// TIA Portal project "LampModel" (V16)

(* hardware
DEVICE "HMI_1"  TP700 Comfort
   slot 0: "HMI_1"  TP700 Comfort  6AV2 124-0GC01-0AX0  16.0.0.0
   slot 1: "HMI_RT_1"  TP700 Comfort  6AV2 124-0GC01-0AX0  16.0.0.0
   slot 5: "HMI_1.IE_CP_1"  PROFINET Interface  16.0.0.0
      slot 1: "PROFINET Interface_1"  PROFINET Interface
         slot 1: "Port_1"  Port
         slot 2: "Port_2"  Port
   slot 7: "HMI_1.MPI/DP_CP_1"  MPI/DP Interface  16.0.0.0
DEVICE "S71500/ET200MP station_1"  S7-1500 station
   slot 0: "Rail_0"  Rack  6ES7 590-1***0-0AA0
   slot 1: "PLC_1"  CPU 1518-4 PN/DP  6ES7 518-4AP00-0AB0  V2.8
      slot 3: "CPU display_1"  6ES7591-1BA00-0AA0
      slot 32768: "PROFINET interface_1"  X1
         slot 32769: "Port_1"  X1 P1
         slot 32770: "Port_2"  X1 P2
      slot 33024: "PROFINET interface_2"  X2
         slot 33025: "Port_1"  X2 P1
      slot 33280: "PROFINET interface GBIT_3"  X3
         slot 33281: "Port_1"  X3 P1
      slot 33536: "DP interface_1"  X4
      slot 34817: "Virtual CP interface port_1"  Virtual CP interface port  Virtual CP interface port
*)

// ===== PLC "PLC_1"  CPU 1518-4 PN/DP =====

VAR_GLOBAL   // PLC tag table "Default tag table"
   "Lambayı Yak" AT %M0.0 : Bool;
   "Lamba" AT %M0.1 : Bool;
   "PTRIG" AT %M0.2 : Bool;
   "PTRIG1" AT %M0.3 : Bool;
   "NTRIG" AT %M0.4 : Bool;
   "PTRIG3" AT %M0.5 : Bool;
   "ntrıg2" AT %M0.6 : Bool;
END_VAR

ORGANIZATION_BLOCK "Main"   // OB1, LAD, ProgramCycle
TITLE = "Main Program Sweep (Cycle)"
{ S7_Optimized_Access := 'TRUE' }
VERSION : 0.1
   VAR_INPUT
      Initial_Call : Bool;   // Initial call of this OB
      Remanence : Bool;   // =True, if remanent data are available
   END_VAR
   VAR_TEMP   // added for the SCL form of the ladder/FBD networks
      _w1 : Bool;
      _w2 : Bool;
   END_VAR
BEGIN

REGION Network 1
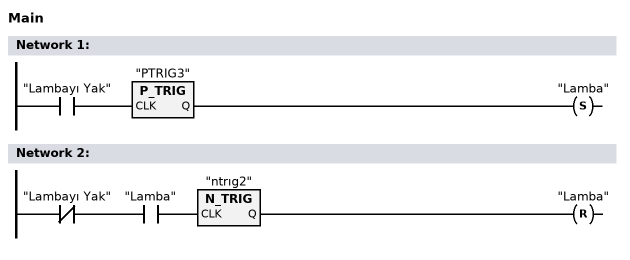
   RUNG wire#powerrail
      Contact( "Lambayı Yak" )
      P_Trig( "PTRIG3" )
      S_Coil( "Lamba" )
   END_RUNG
   // the same network as SCL:
   #_w1 := "Lambayı Yak" AND NOT "PTRIG3";   // rising edge
   "PTRIG3" := "Lambayı Yak";
   IF #_w1 THEN "Lamba" := TRUE; END_IF;
END_REGION

REGION Network 2
   RUNG wire#powerrail
      I_Contact( "Lambayı Yak" )
      Contact( "Lamba" )
      N_Trig( "ntrıg2" )
      R_Coil( "Lamba" )
   END_RUNG
   // the same network as SCL:
   #_w1 := NOT "Lambayı Yak" AND "Lamba";
   #_w2 := NOT #_w1 AND "ntrıg2";   // falling edge
   "ntrıg2" := #_w1;
   IF #_w2 THEN "Lamba" := FALSE; END_IF;
END_REGION
END_ORGANIZATION_BLOCK

(* ===== HMI "HMI_RT_1" =====
system functions are stored by id; their names below are inferred from use
connection "HMI_Connection_1": ETHERNET, S7_1500_OMS

HMI tags "Default tag table"
   "Tag_ScreenNumber" : UInt, internal
   "Lambayı Yak" : Bool = PLC "Lambayı Yak" AT %M0.0, 1 s
   "Lamba" : Bool = PLC Lamba AT %M0.1, 1 s

screen "Root screen" 800x420, template "Template_1"
   Button "Button_1" at 167,146 size 188x32; TextOff 'Lambayı Yak'
      on Press: function_b14e0dd5("Lambayı Yak", 0)
      Appearance <- "Lambayı Yak"
   GraphicView "Graphic view_2" at 454,108 size 77x98; Picture "Graphic_2"
      Appearance <- "Lambayı Yak"
   Circle "Circle_1" at 592,146 size 48x48
      Appearance <- "Lamba"

Template "Template_1" 800x420
   Button "Exit" at 720,360 size 78x58; TextOff 'Exit'; PictureOff "ExitRuntime_TP700_Comfort_TR"; PictureOn "ExitRuntime_TP700_Comfort_TR"
      on Release: StopRuntime(0)
   Button "Template_Button" at 640,360 size 78x58; TextOff 'Text'
   Button "Template_Button_1" at 560,360 size 78x58; TextOff 'Text'
   Button "Template_Button_2" at 480,360 size 78x58; TextOff 'Text'
   Button "Template_Button_3" at 400,360 size 78x58; TextOff 'Text'
   Button "Template_Button_4" at 321,360 size 78x58; TextOff 'Text'
   Button "Template_Button_5" at 241,360 size 78x58; TextOff 'Text'
   Button "Template_Button_6" at 161,360 size 78x58; TextOff 'Text'
   Button "Template_Button_7" at 81,360 size 78x58; TextOff 'Text'
   Button "Start screen" at 1,360 size 78x58; TextOff 'Start screen'; PictureOff "NavigateHome_TP700_Comfort_TR"; PictureOn "NavigateHome_TP700_Comfort_TR"
      on Release: ActivateScreen("Root screen", 0)
*)